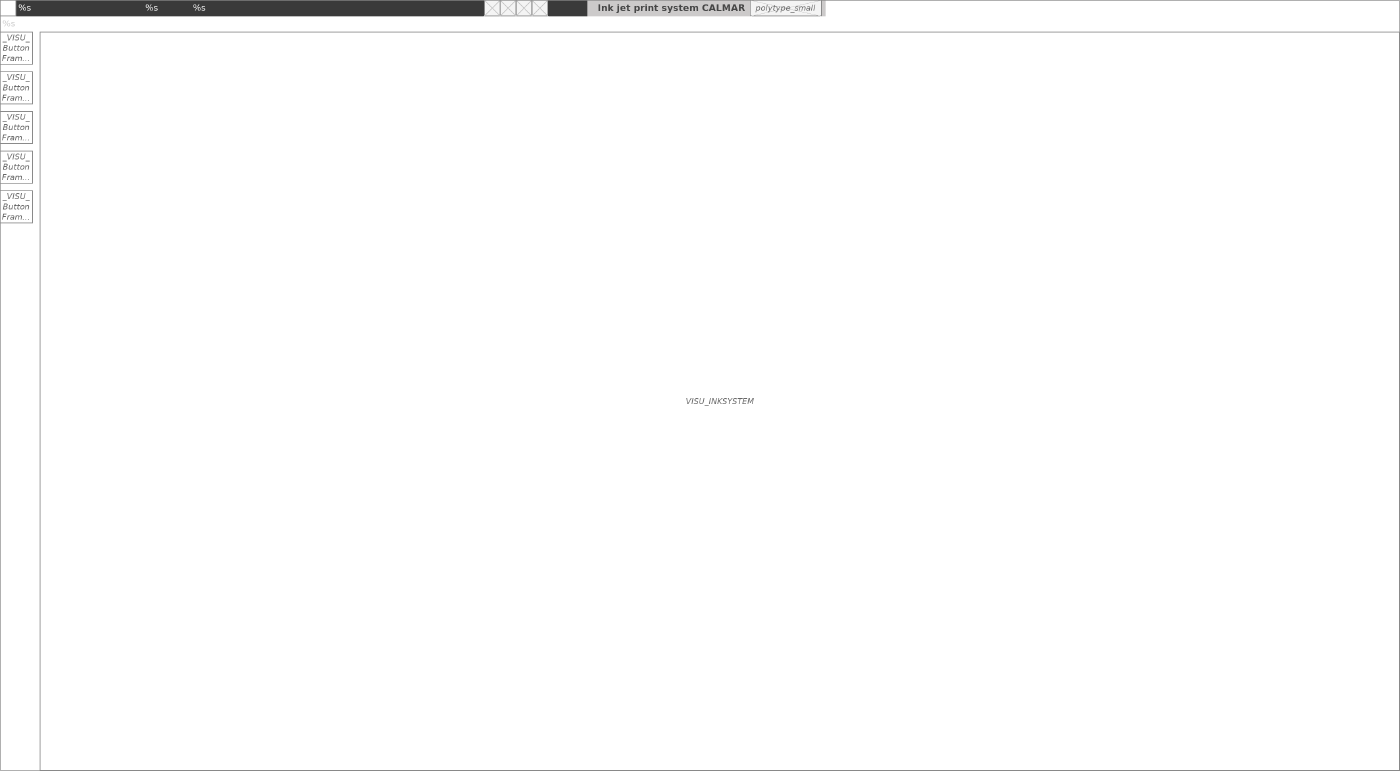
VISUALIZATION VISU_Main  // 1764x972
    Frame (50,40 1714x932), frame switch variable: PRG_SYSTEM.nMainVisuFrameIndex
        shows VISU_INKSYSTEM()
        shows VISU_PrintOverview()
        shows CalmarCompSystem.VISU_RECIPE()
        shows VISU_SERVICE()
        shows VISU_MACHINE()
    Frame (0,40 41x41)
        shows _VISU_ButtonFrameSel(mCfg := PRG_SYSTEM.sMainButtons[0])
    Rectangle (0,20 200x20), "%s", text variable: PRG_SYSTEM.sMainButtons[PRG_SYSTEM.nMainVisuFrameIndex].sVisuName
    Group (20,0 1020x20)
        Rectangle (0,0 1020x20)
        Rectangle (0,0 160x20), "%s", text variable: PRG_SYSTEM.sC_Ads_System.aProject
        Rectangle (160,0 60x20), "%s", text variable: PRG_SYSTEM.sC_Ads_System.aMachine
        Rectangle (220,0 120x20), "%s", text variable: PRG_SYSTEM.aCurrentDateTime
        Image (650,0 20x20), invisible if: NOT PRG_MACHINE.bO_ErrorMsgActive, image: GlobalImagePool.error_icon
        Image (610,0 20x20), invisible if: NOT PRG_MACHINE.sO_SystemCmd.bEStop, image: GlobalImagePool.estop_icon
        Image (590,0 20x20), invisible if: NOT PRG_MACHINE.sO_SystemCmd.bSleep, image: GlobalImagePool.sleep_icon
        Image (630,0 20x20), invisible if: NOT PRG_MACHINE.bO_WarningMsgActive, image: GlobalImagePool.warning_icon
        Rectangle (720,0 300x20)
        Image (925,0 90x20), image: polytype_small
        Rectangle (730,0 200x20), "Ink jet print system CALMAR"
    Frame (0,90 41x41)
        shows _VISU_ButtonFrameSel(mCfg := PRG_SYSTEM.sMainButtons[1])
    Frame (0,140 41x41)
        shows _VISU_ButtonFrameSel(mCfg := PRG_SYSTEM.sMainButtons[2])
    Frame (0,190 41x41)
        shows _VISU_ButtonFrameSel(mCfg := PRG_SYSTEM.sMainButtons[3])
    Frame (0,0 20x20)
        shows VISU_ButtonHome()
    Frame (0,240 41x41)
        shows _VISU_ButtonFrameSel(mCfg := PRG_SYSTEM.sMainButtons[4])
END_VISUALIZATION

(* stored: Version 1.1.0.1, ProductVersion 3.1.4024.11
   Visu VISU_Main: Id {4370c45a-c948-45d6-8aa9-b0f4ad4e0f04} *)
